// TIA Portal V15.1 export
// export: Created 2026-01-09T13:45:15.3715696Z, ExportSetting WithDefaults, WithReadOnly, DisplayName Totally Integrated Automation Portal, DisplayVersion V15.1 Update 8, DisplayName TIA Portal Openness, DisplayVersion V15.1 Update 8, DisplayName STEP 7 Professional, DisplayVersion V15.1 Update 8, DisplayName WinCC Advanced, DisplayVersion V15.1 Update 8
FUNCTION "FCCA_CCD_FD1" : Void   // FC12, LAD
{ S7_Optimized_Access := 'TRUE' }
VERSION : 0.1
// stored: AutoNumber true, CodeModifiedDate 2026-01-04T14:27:04.612364Z, CompileDate 2026-01-04T14:27:05.6125141Z, CreationDate 2024-10-13T15:07:34.9617085Z, HandleErrorsWithinBlock false, InterfaceModifiedDate 2024-08-08T03:19:31.8063857Z, IsConsistent true, IsIECCheckEnabled false, IsKnowHowProtected false, IsWriteProtected false, LibraryConformanceStatus Error: The block contains calls of single instances. Warning: The object contains access to global data blocks. Warning: The block contains direct access to inputs, outputs, bit memories, indirect access to the registry or indirect access to external memory areas that are unknown at the time of compilation., ModifiedDate 2026-01-04T14:27:04.612364Z, ParameterModified 2024-08-08T03:19:31.8063857Z, PLCSimAdvancedSupport false, SetENOAutomatically False, StructureModified 2024-08-08T03:19:31.8063857Z, UDAEnableTagReadback false
   VAR_TEMP   // added for the SCL form of the ladder/FBD networks
      _w1 : Bool;
   END_VAR
BEGIN

REGION Network 1: CAN XI MANG 1
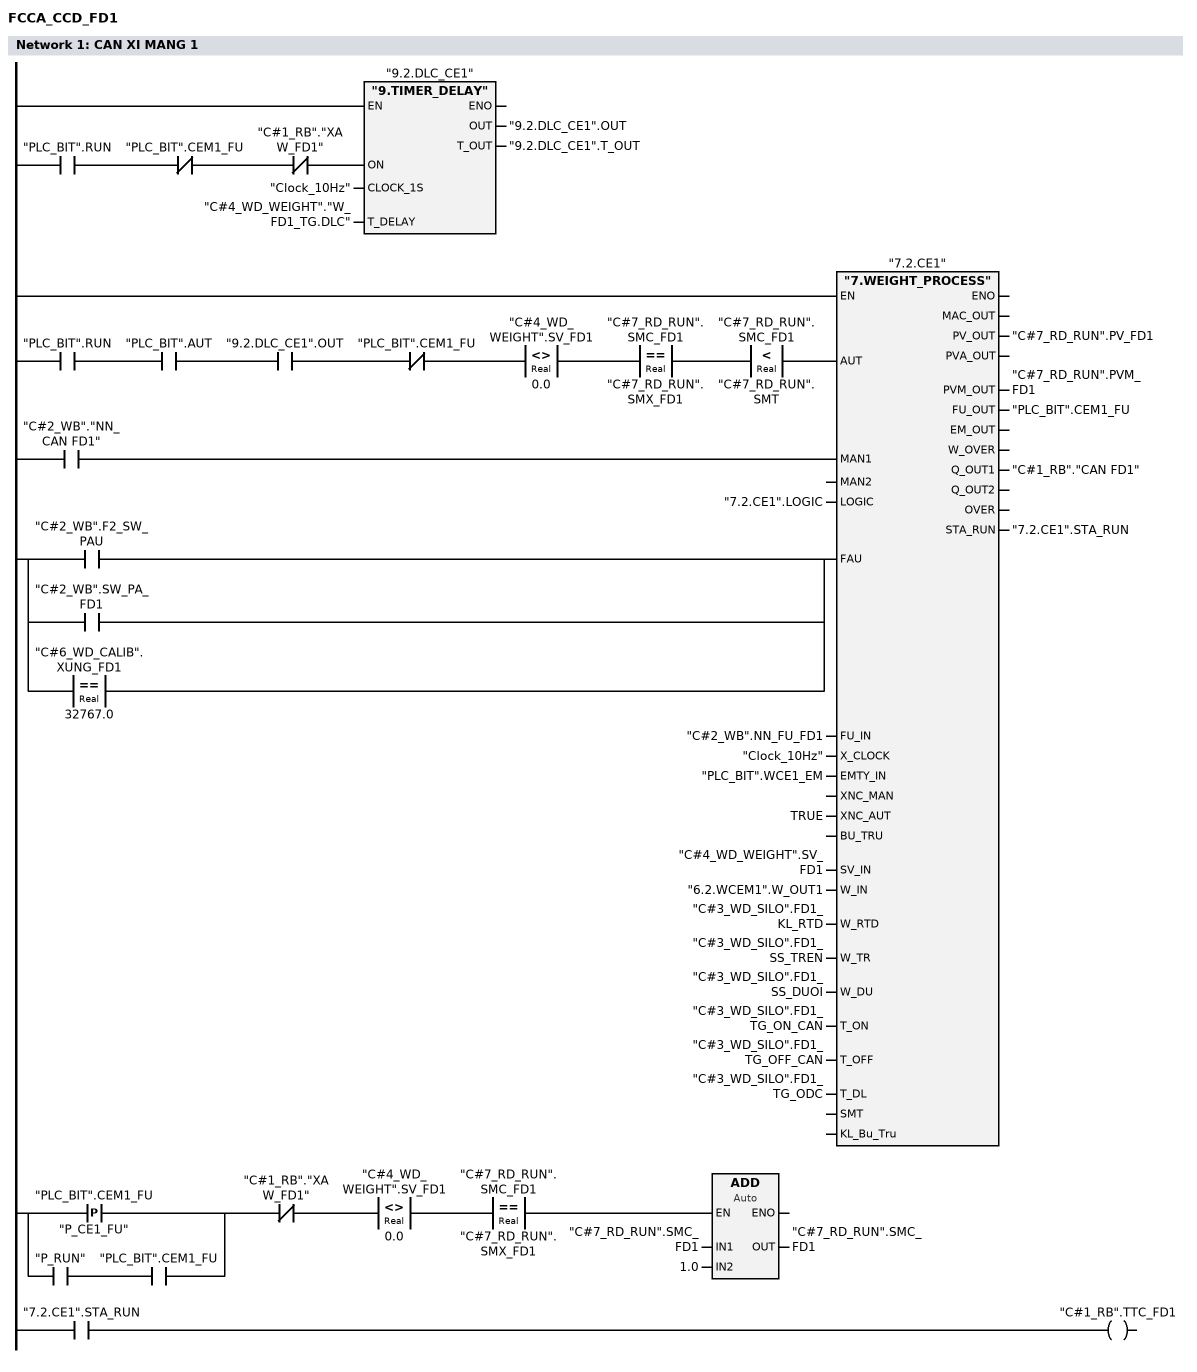
   RUNG wire#powerrail
      "9.2.DLC_CE1"(ON := wire#w1, CLOCK_1S := "Clock_10Hz", T_DELAY := "C#4_WD_WEIGHT"."W_FD1_TG.DLC", OUT => "9.2.DLC_CE1".OUT, T_OUT => "9.2.DLC_CE1".T_OUT)
   END_RUNG
   RUNG wire#powerrail
      Contact( "PLC_BIT".RUN )
      I_Contact( "PLC_BIT".CEM1_FU )
      I_Contact( "C#1_RB"."XA W_FD1" )
   END_RUNG wire#w1
   RUNG wire#powerrail
      "7.2.CE1"(AUT := wire#w2, MAN1 := wire#w3, FAU := wire#w4, MAN2 :=, LOGIC := "7.2.CE1".LOGIC, FU_IN := "C#2_WB".NN_FU_FD1, X_CLOCK := "Clock_10Hz", EMTY_IN := "PLC_BIT".WCE1_EM, XNC_MAN :=, XNC_AUT := TRUE, BU_TRU :=, SV_IN := "C#4_WD_WEIGHT".SV_FD1, W_IN := "6.2.WCEM1".W_OUT1, W_RTD := "C#3_WD_SILO".FD1_KL_RTD, W_TR := "C#3_WD_SILO".FD1_SS_TREN, W_DU := "C#3_WD_SILO".FD1_SS_DUOI, T_ON := "C#3_WD_SILO".FD1_TG_ON_CAN, T_OFF := "C#3_WD_SILO".FD1_TG_OFF_CAN, T_DL := "C#3_WD_SILO".FD1_TG_ODC, SMT :=, KL_Bu_Tru :=, MAC_OUT =>, PV_OUT => "C#7_RD_RUN".PV_FD1, PVA_OUT =>, PVM_OUT => "C#7_RD_RUN".PVM_FD1, FU_OUT => "PLC_BIT".CEM1_FU, EM_OUT =>, W_OVER =>, Q_OUT1 => "C#1_RB"."CAN FD1", Q_OUT2 =>, OVER =>, STA_RUN => "7.2.CE1".STA_RUN)
   END_RUNG
   RUNG wire#powerrail
      Contact( "PLC_BIT".RUN )
      Contact( "PLC_BIT".AUT )
      Contact( "9.2.DLC_CE1".OUT )
      I_Contact( "PLC_BIT".CEM1_FU )
      { S7_Templates := "SrcType := Real" } NE_Contact(in1 := "C#4_WD_WEIGHT".SV_FD1, in2 := 0.0)
      { S7_Templates := "SrcType := Real" } EQ_Contact(in1 := "C#7_RD_RUN".SMC_FD1, in2 := "C#7_RD_RUN".SMX_FD1)
      { S7_Templates := "SrcType := Real" } LT_Contact(in1 := "C#7_RD_RUN".SMC_FD1, in2 := "C#7_RD_RUN".SMT)
   END_RUNG wire#w2
   RUNG wire#powerrail
      Contact( "C#2_WB"."NN_CAN FD1" )
   END_RUNG wire#w3
   RUNG wire#powerrail
      Contact( "C#2_WB".F2_SW_PAU )
   END_RUNG wire#w4
   RUNG wire#powerrail
      Contact( "C#2_WB".SW_PA_FD1 )
   END_RUNG wire#w4
   RUNG wire#powerrail
      { S7_Templates := "SrcType := Real" } EQ_Contact(in1 := "C#6_WD_CALIB".XUNG_FD1, in2 := 32767.0)
   END_RUNG wire#w4
   RUNG wire#powerrail
      P_Contact(operand := "PLC_BIT".CEM1_FU, bit := "P_CE1_FU")
      wire#w5
      I_Contact( "C#1_RB"."XA W_FD1" )
      { S7_Templates := "SrcType := Real" } NE_Contact(in1 := "C#4_WD_WEIGHT".SV_FD1, in2 := 0.0)
      { S7_Templates := "SrcType := Real" } EQ_Contact(in1 := "C#7_RD_RUN".SMC_FD1, in2 := "C#7_RD_RUN".SMX_FD1)
      Add(in1 := "C#7_RD_RUN".SMC_FD1, in2 := 1.0, out => "C#7_RD_RUN".SMC_FD1)
   END_RUNG
   RUNG wire#powerrail
      Contact( "P_RUN" )
      Contact( "PLC_BIT".CEM1_FU )
   END_RUNG wire#w5
   RUNG wire#powerrail
      Contact( "7.2.CE1".STA_RUN )
      Coil( "C#1_RB".TTC_FD1 )
   END_RUNG
   // the same network as SCL:
   "9.2.DLC_CE1"(ON := "PLC_BIT".RUN AND NOT "PLC_BIT".CEM1_FU AND NOT "C#1_RB"."XA W_FD1",   // "9.TIMER_DELAY"
                 CLOCK_1S := "Clock_10Hz",
                 T_DELAY := "C#4_WD_WEIGHT"."W_FD1_TG.DLC",
                 OUT => "9.2.DLC_CE1".OUT,
                 T_OUT => "9.2.DLC_CE1".T_OUT);
   "7.2.CE1"(AUT := "PLC_BIT".RUN AND "PLC_BIT".AUT AND "9.2.DLC_CE1".OUT AND NOT "PLC_BIT".CEM1_FU AND ("C#4_WD_WEIGHT".SV_FD1 <> 0.0) AND ("C#7_RD_RUN".SMC_FD1 = "C#7_RD_RUN".SMX_FD1) AND ("C#7_RD_RUN".SMC_FD1 < "C#7_RD_RUN".SMT),   // "7.WEIGHT_PROCESS"
             MAN1 := "C#2_WB"."NN_CAN FD1",
             LOGIC := "7.2.CE1".LOGIC,
             FAU := "C#2_WB".F2_SW_PAU OR "C#2_WB".SW_PA_FD1 OR ("C#6_WD_CALIB".XUNG_FD1 = 32767.0),
             FU_IN := "C#2_WB".NN_FU_FD1,
             X_CLOCK := "Clock_10Hz",
             EMTY_IN := "PLC_BIT".WCE1_EM,
             XNC_AUT := TRUE,
             SV_IN := "C#4_WD_WEIGHT".SV_FD1,
             W_IN := "6.2.WCEM1".W_OUT1,
             W_RTD := "C#3_WD_SILO".FD1_KL_RTD,
             W_TR := "C#3_WD_SILO".FD1_SS_TREN,
             W_DU := "C#3_WD_SILO".FD1_SS_DUOI,
             T_ON := "C#3_WD_SILO".FD1_TG_ON_CAN,
             T_OFF := "C#3_WD_SILO".FD1_TG_OFF_CAN,
             T_DL := "C#3_WD_SILO".FD1_TG_ODC,
             PV_OUT => "C#7_RD_RUN".PV_FD1,
             PVM_OUT => "C#7_RD_RUN".PVM_FD1,
             FU_OUT => "PLC_BIT".CEM1_FU,
             Q_OUT1 => "C#1_RB"."CAN FD1",
             STA_RUN => "7.2.CE1".STA_RUN);
   #_w1 := "PLC_BIT".CEM1_FU AND NOT "P_CE1_FU";   // rising edge of "PLC_BIT".CEM1_FU
   "P_CE1_FU" := "PLC_BIT".CEM1_FU;
   IF (#_w1 OR ("P_RUN" AND "PLC_BIT".CEM1_FU)) AND NOT "C#1_RB"."XA W_FD1" AND ("C#4_WD_WEIGHT".SV_FD1 <> 0.0) AND ("C#7_RD_RUN".SMC_FD1 = "C#7_RD_RUN".SMX_FD1) THEN
       "C#7_RD_RUN".SMC_FD1 := "C#7_RD_RUN".SMC_FD1 + 1.0;
   END_IF;
   "C#1_RB".TTC_FD1 := "7.2.CE1".STA_RUN;
END_REGION
END_FUNCTION
